// TIA Portal V16 export
// export: Created 2024-03-27T10:00:41.8778248Z, ExportSetting WithDefaults, DisplayName Totally Integrated Automation Portal, DisplayVersion V16, DisplayName TIA Portal Version Control Interface, DisplayVersion V16, DisplayName TIA Portal Openness, DisplayVersion V16, DisplayName STEP 7 Professional, DisplayVersion V16, DisplayName STEP 7 Safety, DisplayVersion V16, DisplayName WinCC Advanced, DisplayVersion V16
TYPE "UR__T2O_Safety"
// stored: IsFailsafeCompliant false
   STRUCT
      "Safety mode" : USInt;
      Reserved_1 { ExternalAccessible := 'False'; ExternalVisible := 'False'; ExternalWritable := 'False'} : USInt;
      Reserved_2 { ExternalAccessible := 'False'; ExternalVisible := 'False'; ExternalWritable := 'False'} : UInt;
      "NO: Is normal mode" : Bool;
      "RD: Is reduced mode" : Bool;
      "PS: Is protective stopped" : Bool;
      "RC: Is recovery mode" : Bool;
      "SS: Is safeguard stopped" : Bool;
      "SES: Is system emergency stopped" : Bool;
      "RES: Is robot emergency stopped" : Bool;
      "ES: Is emergency stopped" : Bool;
      "VL: Is violation" : Bool;
      "FT: Is fault" : Bool;
      "ST: Is stopped due to safety" : Bool;
      Reserved_11 { ExternalAccessible := 'False'; ExternalVisible := 'False'; ExternalWritable := 'False'} : Bool;
      Reserved_12 { ExternalAccessible := 'False'; ExternalVisible := 'False'; ExternalWritable := 'False'} : Bool;
      Reserved_13 { ExternalAccessible := 'False'; ExternalVisible := 'False'; ExternalWritable := 'False'} : Bool;
      Reserved_14 { ExternalAccessible := 'False'; ExternalVisible := 'False'; ExternalWritable := 'False'} : Bool;
      Reserved_15 { ExternalAccessible := 'False'; ExternalVisible := 'False'; ExternalWritable := 'False'} : Bool;
      Reserved_16_31 { ExternalAccessible := 'False'; ExternalVisible := 'False'; ExternalWritable := 'False'} : UInt;
   END_STRUCT;
END_TYPE
